TYPE ST_Machine_Status :
    STRUCT
		PackMLState : E_PMLStateForHMI;
    END_STRUCT
END_TYPE

(* stored: Version 1.1.0.1, ProductVersion 3.1.4024.15
   DUT ST_Machine_Status: Id {d69beaae-0411-481a-a2b6-ca5760b7a431} *)
